FUNCTION_BLOCK TcoTaskTest EXTENDS TcoTask
VAR
	_IsBusy						:	BOOL;	
	_IsError					:	BOOL;	
	_IsDone						:	BOOL;	
	_CounterSetValue			:	ULINT;
	_CounterValue				:	ULINT;
	_InvokeCounter				:	ULINT;
	_ExecuteCounter				:	ULINT;
	_DoneCounter				:	ULINT;	
	_InvokeRisingEdgeCounter	:	ULINT;
	_ExecuteRisingEdgeCounter	:	ULINT;
	_DoneRisingEdgeCounter		:	ULINT;	
	_PreviousState				:	eTaskState;
	_CounterValuePV				:	ULINT;
	_MyIdentity					:	ULINT;
	_MyContextIdentity			:	ULINT;
	_MyContextStartCount 		:	ULINT;
	_MyContextEndCount			:	ULINT;	
	_MyParentIdentity			:	ULINT;
	_AutoRestoreByMyParentEnabled	: BOOL;	
END_VAR

ExecutionBody();

{attribute 'TcRpcEnable'}
METHOD INTERNAL ExecutionBody
IF(THIS^._taskState = eTaskState.Request) THEN
	_InvokeCounter := _InvokeCounter + 1; 
END_IF;

IF(THIS^._taskState = eTaskState.Request AND _PreviousState <> eTaskState.Request) THEN
	_CounterValue	:=	_CounterSetValue;
	_CounterValuePV := _CounterValue;
	_InvokeRisingEdgeCounter := _InvokeRisingEdgeCounter + 1;
END_IF

IF(THIS^._taskState = eTaskState.Executing AND _PreviousState <> eTaskState.Executing) THEN
	_ExecuteRisingEdgeCounter := _ExecuteRisingEdgeCounter + 1;
END_IF

_PreviousState	:=	THIS^._taskState;

IF(Execute()) THEN
	_ExecuteCounter := _ExecuteCounter + 1;	
	_CounterValue := _CounterValue - 1;
	DoneWhen(_CounterValue <= 0);			
	ThrowWhen(ABS(_CounterValuePV -_CounterValue) > 1);
	_CounterValuePV := _CounterValue;
END_IF

IF(THIS^._taskState = eTaskState.Done) THEN
	_DoneCounter := _DoneCounter + 1; 
END_IF;

IF(THIS^._taskState = eTaskState.Done AND _PreviousState <> eTaskState.Done) THEN
	_DoneRisingEdgeCounter := _DoneRisingEdgeCounter + 1; 
END_IF
END_METHOD

{attribute 'TcRpcEnable'}
METHOD INTERNAL GetMessage : STRING
GetMessage := SUPER^._messenger._mime.Text;
END_METHOD

{attribute 'TcRpcEnable'}
METHOD INTERNAL PostMessage
VAR_INPUT
	Message	:	STRING;
END_VAR
THIS^.Messenger.Post(Message ,eMessageCategory.Error);
END_METHOD

{attribute 'TcRpcEnable'}
METHOD INTERNAL ReadOutAutoRestoreProperties
_AutoRestoreByMyParentEnabled	:= THIS^.AutoRestorable;
END_METHOD

{attribute 'TcRpcEnable'}
METHOD INTERNAL ReadOutIdentities
_MyIdentity			:=	THIS^.Identity;

_MyContextIdentity	:=	THIS^.Context.Identity;
		
_MyContextStartCount :=	THIS^.Context.StartCycleCount;

_MyContextEndCount	:=	THIS^.Context.EndCycleCount;

_MyParentIdentity	:=	THIS^._Parent.Identity;
END_METHOD

{attribute 'TcRpcEnable'}
METHOD INTERNAL ReadOutState
_IsBusy		:=	THIS^.Busy;	
_IsError	:=	THIS^.Error;	
_IsDone		:=	THIS^.Done;
END_METHOD

{attribute 'TcRpcEnable'}
METHOD INTERNAL SetPreviousStateToIdle
THIS^._PreviousState := eTaskState.Idle;
END_METHOD

{attribute 'TcRpcEnable'}
METHOD INTERNAL TriggerAbort
THIS^.Abort();
END_METHOD

{attribute 'TcRpcEnable'}
METHOD INTERNAL TriggerInvoke
THIS^.Invoke();
END_METHOD

{attribute 'TcRpcEnable'}
METHOD INTERNAL TriggerRestore
THIS^.Restore();
END_METHOD

END_FUNCTION_BLOCK

(* stored: Version 1.1.0.1, ProductVersion 3.1.4024.6
   POU TcoTaskTest: Id {9aa8db61-0cc6-40c6-9397-95033027855c}, SpecialFunc None
   Method ExecutionBody: Id {77a5a45d-9cd7-4d75-83c5-1e7025fc00d2}
   Method GetMessage: Id {8e6f936b-bc35-4ef7-a147-2025c495357f}
   Method PostMessage: Id {5fc16e78-a33a-4b3d-b72e-63dff904b3c2}
   Method ReadOutAutoRestoreProperties: Id {5b83d008-369d-4819-8af0-9c589c21787c}
   Method ReadOutIdentities: Id {97964902-e608-40e8-94bf-85004e67f007}
   Method ReadOutState: Id {8a834a60-c289-4ad1-a649-a06b124cc84a}
   Method SetPreviousStateToIdle: Id {5b4ca5af-515c-4456-914e-015624dcdd9a}
   Method TriggerAbort: Id {fb8d5aab-1b46-4b74-a563-a929ff61965a}
   Method TriggerInvoke: Id {eaf79119-f66d-4e8d-8769-8d600bac760b}
   Method TriggerRestore: Id {bc4db07e-7c8f-4208-80ac-22e04a9c54df} *)
